FUNCTION_BLOCK Tramp
VAR_INPUT
	Dir: INT := -1;
	Strobe: BOOL;
END_VAR
VAR_OUTPUT
END_VAR
VAR
	AtPos: INT;
	Goto_Pos: INT;
	Status: INT := 0;
	Error: BOOL;
	Speed: INT;
	Display : STRING;
END_VAR

IF Strobe THEN
	Goto_Pos := Goto_Pos + dir;
END_IF


GVL.qiAtStation1 := FALSE;
GVL.qiAtStation2 := FALSE;
IF AtPos > -50 AND atPos < 1 THEN
	GVL.qiAtStation1 := TRUE;
	//GVL.qiDisplay:='At Station1';
ELSIF AtPos > 550 AND atPos < 600 THEN
	GVL.qiAtStation2 := TRUE;
	//GVL.qiDisplay:='At Station2';
END_IF

IF AtPos > -40 AND AtPos <600 THEN
	AtPos := Goto_Pos;
	//GVL.qiDisplay:='On the way';
END_IF

END_FUNCTION_BLOCK

(* stored: Version 1.1.0.1, ProductVersion 3.1.4024.12
   POU Tramp: Id {820d301d-2dad-4f98-b113-d2dc72b186e4}, SpecialFunc None *)
